(* Schneider Machine Expert - Basic project Persistent Var, file version 1.8.0.0 *)
(* ProjectInformations: Name=Yeni proje *)

HARDWARE
  Cpu 0: TM221ME16T/G
  ModuleExtensionObject 0: TM3DI8/G
  ModuleExtensionObject 1: TM3AQ2/G
  EthernetConfiguration: NetworkName=M221, IpAllocationMode=FixedAddress, IpAddress=192.168.0.15, SubnetMask=255.255.255.0
  SerialLineConfiguration: Baud=Baud19200, Parity=ParityNone, DataBits=DataBits8, StopBits=StopBits1, PhysicalMedium=PhysicalMediumRs485, TransmissionMode=TransmissionModeModbusRtu, SlaveId=1, Addressing=SlaveAddressing
  MastTask: UsePeriodScanMode=false, PeriodScan=100
  FastTask: Period=255
  CpuBehavior: StartingMode=StartAsPreviousState, AutoSaveRamOnEeprom=true, WatchdogPeriod=250

SYMBOLS  (address, symbol, comment, settings)
  %M0         "HMI/FIRÇA YUKARI"
  %M1         "HMI/FIRÇA AŞAĞI"
  %M2         "HMI/FIRÇA 2 YUKARI"
  %M3         "HMI/FIRÇA 2 AŞAĞI"
  %M4         "HMI BANT START"
  %M5         "HMI OSILASYON START"
  %M6         "427/FIRCA INVERTOR"
  %M7         "428/VALF"
  %M8         "STOP"
  %M10        "ENC 1 PRESET"
  %M11        "ENC 2 PRESET"
  %M12        "ENC_1_SIFIRLAMA"
  %M13        "ENC_2_SIFIRLAMA"
  %M49        "ENCODER ENABLE"
  %S93      SB_MWBACKUP  "User set this bit to 1 to store the %MW variable in the flash (up to 2000)"
  %S94      SB_MWRESTORE  "User set this bit to 1 to restore the saved data"
  %SW148    SW_NBPERS  "Number of persistent variables (maximum 2000)"
  %C0         "HAFIZADAN ENKODERLERİ ÇEK"
  %R0         "ENKODER 1 HAFIZAYA AT"  [Type=Lifo]
  %R1         "ENKODER 2 HAFIZAYA AT"  [Type=Lifo]
  %I0.0       "403/FIRÇA1 ÜST SINIR ANAHTARI"
  %I0.1       "402/FIRÇA1 ALT SINIR ANAHTARI"
  %I0.2       "405/FIRÇA2/ÜST SINIR ANAHTARI"
  %I0.3       "404/FIRÇA2/ ALT SINIR ANAHTARI"
  %Q0.0       "421/FIRÇA YUKARI"
  %Q0.1       "422/FIRÇA AŞAĞI"
  %Q0.2       "423/FIRÇA 2 YUKARI"
  %Q0.3       "424/FIRÇA 2 AŞAĞI"
  %Q0.4       "425/BANT START"
  %Q0.5       "426/OSILASYON START"
  %Q0.6       "427/FIRCA INVERTER"
  %Q0.7       "428/VALF"
  %HSC0       "FIRÇA1/ENKODER"  [Type=CounterOrDownCounterBiPhasesX1, Preset=0, DedicatedInputs(DedicatedInput(Activated=true), DedicatedInput(Activated=true)), ReflexOutputs(ReflexOutput(Activated=false, LessThanS0=false, GreaterOrEqualThanS0=false, GreaterOrEqualThanS1=false), ReflexOutput(Activated=false, LessThanS0=false, GreaterOrEqualThanS0=false, GreaterOrEqualThanS1=false)), Thresholds(Threshold(ThresholdType=NotUsed, Pri]
  %HSC1       "FIRÇA2/ENKODER"  [Type=CounterOrDownCounterBiPhasesX1, Preset=0, DedicatedInputs(DedicatedInput(Activated=true), DedicatedInput(Activated=true)), ReflexOutputs(ReflexOutput(Activated=false, LessThanS0=false, GreaterOrEqualThanS0=false, GreaterOrEqualThanS1=false), ReflexOutput(Activated=false, LessThanS0=false, GreaterOrEqualThanS0=false, GreaterOrEqualThanS1=false)), Thresholds(Threshold(ThresholdType=NotUsed, Pri]
  %I1.0       "403/FIRÇA UST SINIR SWITCH"
  %I1.1       "402/FIRÇA ALT SINIR SWITCH"
  %I1.2       "405/FIRÇA2/ÜST SINIR SWITCH"
  %I1.3       "404/FIRÇA2/ALT SINIR SWITCH"

POU Yeni POU
  (* SectionNumber=1 *)

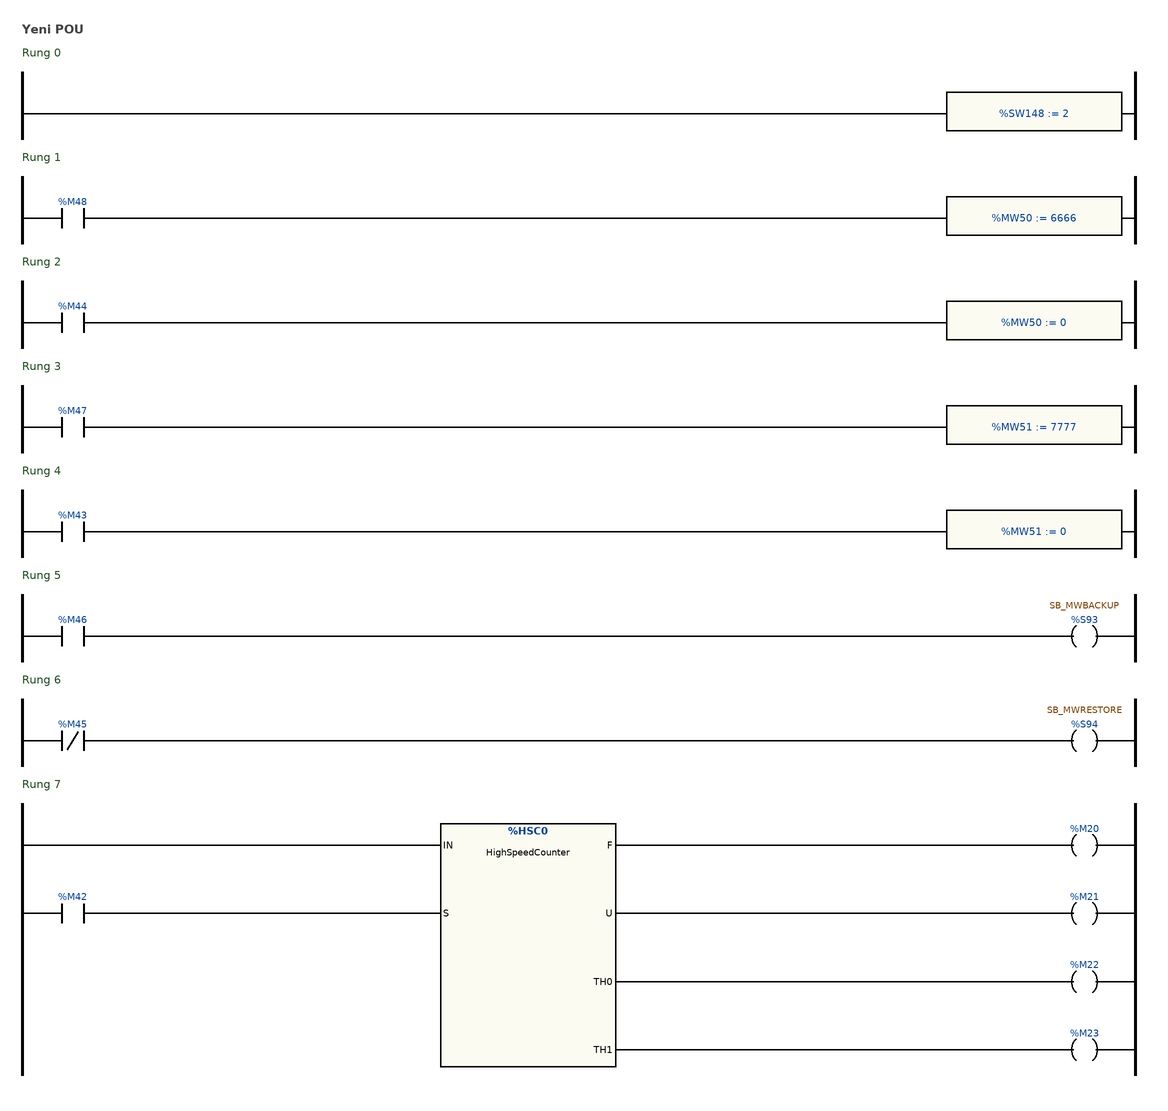

// Rung 0
  LD 1
  [ %SW148 := 2 ]         (* SW_NBPERS *)
  // as ST:
  //   SW_NBPERS := 2;

// Rung 1
  LD %M48
  [ %MW50 := 6666 ]
  // as ST:
  //   IF %M48 THEN %MW50 := 6666; END_IF;

// Rung 2
  LD %M44
  [ %MW50 := 0 ]
  // as ST:
  //   IF %M44 THEN %MW50 := 0; END_IF;

// Rung 3
  LD %M47
  [ %MW51 := 7777 ]
  // as ST:
  //   IF %M47 THEN %MW51 := 7777; END_IF;

// Rung 4
  LD %M43
  [ %MW51 := 0 ]
  // as ST:
  //   IF %M43 THEN %MW51 := 0; END_IF;

// Rung 5
  LD %M46
  ST %S93                 (* SB_MWBACKUP *)
  // as ST:
  //   SB_MWBACKUP := %M46;

// Rung 6
  LDN %M45
  ST %S94                 (* SB_MWRESTORE *)
  // as ST:
  //   SB_MWRESTORE := NOT %M45;

// Rung 7
  BLK %HSC0
  LD 1
  IN
  LD %M42
  S
  OUT_BLK
  LD F
  ST %M20
  LD U
  ST %M21
  LD TH0
  ST %M22
  LD TH1
  ST %M23
  END_BLK
  // as ST:
  //   %HSC0(IN := TRUE, S := %M42);
  //   %M20 := %HSC0.F;
  //   %M21 := %HSC0.U;
  //   %M22 := %HSC0.TH0;
  //   %M23 := %HSC0.TH1;

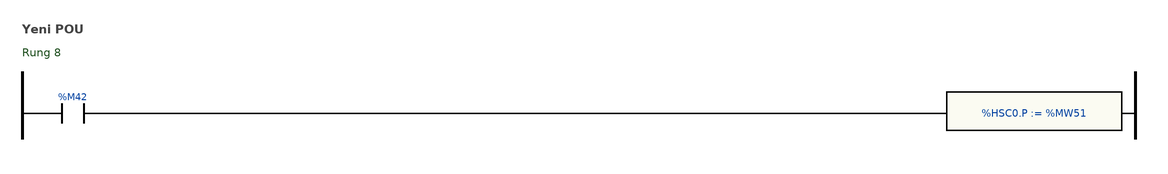

// Rung 8
  LD %M42
  [ %HSC0.P := %MW51 ]
  // as ST:
  //   IF %M42 THEN %HSC0.P := %MW51; END_IF;
